{attribute 'qualified_only'}
VAR_GLOBAL
	// Motion Ref
	// Sine Parameters
	fAmplitude 	: LREAL := 0.1;
	fMean 		: LREAL := 0.2;
	fFrequency 	: LREAL := 0.05;
	
	
	// Valve Values
	// Flow
	fQMaxDown 	: LREAL := 15.9; // [L/min]
	fQMaxUp 	: LREAL := 24.4; // [L/min]	
	
	// Area
	fAreaUp 	: LREAL := 33.100/1E4; //[mm^2]
	fAreaDown 	: LREAL := 23.560/1E4; //[mm^2]
	
	// Deadband
	fDeadUp : LREAL := 0.13;
	fDeadDown : LREAL := 0.13;
	
	fMaxSpeed : LREAL := 0.01; // [m/s] 
	fDeltaP0 : LREAL := 8; // [Bar]
	
	// Deadband test
	fConst : LREAL := 0.0; // [-1, 1]

	fCycleTime : LREAL := 0.001; // Time Step [s]
	fQConst : LREAL := 15;
	
	// PID-constants
	Kp : LREAL := 14.0; 	// P
	Ki : LREAL := 0.0;		// I
	Kd : LREAL := 0.0;		// D
	
	
	
	
END_VAR

(* stored: Version 1.1.0.1, ProductVersion 3.1.4024.12
   GVL G_Parameter: Id {6529201b-0264-4389-a4a9-6a2e97edbca5} *)
